(* CODESYS project Jacomex.project

Project tree, tasks and I/O mapping:
  IIoT_MQTT : XV300, Eaton Automation, version 3.5.19.30
    application Application
      libraries: StringUtils, 3.5.18.0 (System); VisuDialogs, * (System); Web Socket Client SL, 1.9.0.0 (CODESYS); Net Base Services, 3.5.19.20 (3S - Smart Software Solutions GmbH); MQTT Client SL, 1.9.0.0 (CODESYS); Standard, 3.5.18.0 (System); SysTimeRtc, * (System); SysTypes2 Interfaces, * (System)
      task MainTask (cyclic, interval t#20ms, priority 1) calls PRG
      program PRG [CFC]
      visualisation Visualization
      text list QoSTextlist
      function TerminateString [ST]
      image pool ImagePool
      text list ModeTextList
      text list VersionTextList
      global variables GVL_MQTT
      function FC_DataInMessageContainer [ST]
      data type ReactorType
  text list GlobalTextList
  5ce3da45-db07-42e7-a21c-a00fff4ed8f6|C:\Users\a.werner\Documents\background.jpg
  5ce3da45-db07-42e7-a21c-a00fff4ed8f6|C:\Users\a.werner\Documents\background.jpg
*)

// IIoT_MQTT/Application/ReactorType
{attribute 'qualified_only'}
TYPE ReactorType :
(
	O2 		:= 1,
	H2O 	:= 2,
	Both 	:= 3
)BYTE;
END_TYPE

// IIoT_MQTT/Application/GVL_MQTT
VAR_GLOBAL
	aValueData		:	ARRAY[1..20] OF DINT;		// Value data to transmit
	aTextData		:	ARRAY[1..20] OF STRING;		// Text data to transmit
	aBoolData		:	ARRAY[1..100] OF BOOL;		// Boolean data to transmit (Settings/Alarms/Triggers)
END_VAR

// IIoT_MQTT/Application/PRG
// MQTT Client with visualization
PROGRAM PRG
VAR
	//mqttClient 				: MQTT.MQTTClient; 								// Function block to establish a connection to a MQTT broker
	mqttPublisher 			: MQTT.MQTTPublish; 							// Function block to publish MQTT messages
	mqttPublisher2 			: MQTT.MQTTPublish; 							// Function block to publish MQTT messages
	mqttSubscriber 			: MQTT.MQTTSubscribe; 							// Function block to subscribe MQTT topics
	mqttSubscriber2 		: MQTT.MQTTSubscribe; 							// Function block to subscribe MQTT topics
	sHostname 				: STRING(255) 	:= 'mqtts-jacomex.ingelink.dev';//'broker.hivemq.com'; 				// Hostname or ip address or URL (for WebSockets: ws:// or wss://)
	wsUsername				: WSTRING 		:= "wildcard0";
	wsPassword				: WSTRING 		:= "f6eec544dc19429";
	uiPort 					: UINT 			:= 42226; 						// Port of the MQTT broker
	wsPublishTopic 			: WSTRING(1024) := "poly/in/1/0/5169/data"; 							// Topic to publish a message
	wsPublishTopic2 		: WSTRING(1024) := ""; 							// Topic to publish a message
	sWillMessage 			: STRING(1024); 								// The last will message
	abyPublishMessage 		: ARRAY [1..28] OF BYTE; 						// The messsage to publish
	sPublishMessage2 		: STRING(1024) := ''; 							// The messsage to publish 
	rsPub1Error				: RS; 											// Helper to publisher state
	rsPub1Done				: RS; 											// Helper to publisher state
	rsPub2Error				: RS; 											// Helper to publisher state
	rsPub2Done				: RS; 											// Helper to publisher state
	eCommunicationMode 		: MQTT.COMMUNICATION_MODE := MQTT.COMMUNICATION_MODE.TCP; // Communication mode: TCP/IP or WebSockets
	eMQTTVersion 			: MQTT.MQTT_VERSION := MQTT.MQTT_VERSION.V3_1_1; // The MQTT protocol version
	uiKeepAlive				: UINT 		:= 60;	
	sClientID				: STRING 	:= 'wildcard0';
	xCleanSession			: BOOL 		:= TRUE;
	

	
	// If you want to use client certificates, you can configure the connection via the TLS context.	
	 _sCommonName : STRING := 'MyXV303'; // CN of the certificate (common name). 
	 _sCipherList : NBS.CIPHER_LIST := STRUCT(psList := ADR('HIGH'), udiSize := 5); // Cipher string see https://www.openssl.org/docs/man1.1.1/man1/ciphers.html
	 _ciDefaultCertInfo : NBS.CERT_INFO := (psInfo := ADR(_sCommonName), udiSize := SIZEOF(_sCommonName)); // CN of the certificate (common name)

	 _tlsContext : NBS.TLSContext := (	sUseCaseName := _sCommonName, // A certificate is stored in the certificate store with the use case name. You can choose any name. Here we use the common name.
										ePurpose := NBS.PURPOSE.CLIENT_SIDE, // For client certificates set this to NBS.PURPOSE.CLIENT_SIDE
										sTLSVersion := '1.2', // The TLS version
										sCipherList := _sCipherList, // Set the cipher list
										udiVerificationMode := 1, // 2 => Active Peer verification
										ciCertInfo := _ciDefaultCertInfo, // Set the cert info
										itfCertVerifer := 0); // 0 => No Verifier 
	 
	 mqttClient : MQTT.MQTTClient := (itfTLSCOntext := _tlsContext);
    //
	// You can use the method TLSContext.SetInitialValue to set the context while runtime and set the context via the input itfTLSCOntext of the client FB.
	
	dwUuid: DWORD:= 5169;
	xFillingSolenoidValve: BOOL:=TRUE;
	wOxygenValue: WORD := 1664;
	sProject: STRING(16) := 'Project';
	eReactorType: ReactorType:= ReactorType.Both;
END_VAR
VAR // added by the converter: edge detectors and wires of the graphical bodies
    _w1 : ANY;
END_VAR

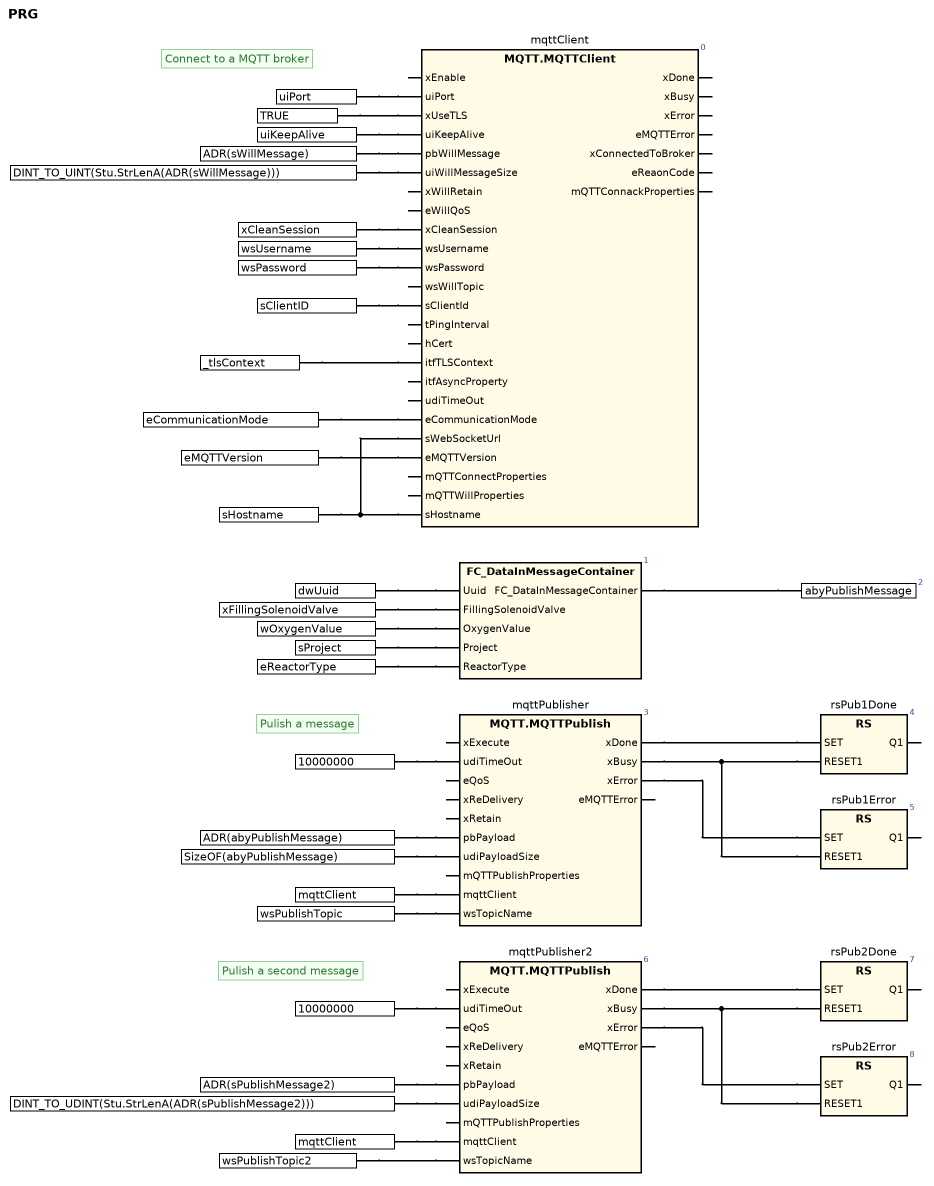
// Connect to a MQTT broker
mqttClient(
    uiPort := uiPort,
    xUseTLS := TRUE,
    uiKeepAlive := uiKeepAlive,
    pbWillMessage := ADR(sWillMessage),
    uiWillMessageSize := DINT_TO_UINT(Stu.StrLenA(ADR(sWillMessage))),
    xCleanSession := xCleanSession,
    wsUsername := wsUsername,
    wsPassword := wsPassword,
    sClientId := sClientID,
    itfTLSContext := _tlsContext,
    eCommunicationMode := eCommunicationMode,
    sWebSocketUrl := sHostname,
    eMQTTVersion := eMQTTVersion,
    sHostname := sHostname); // MQTT.MQTTClient
_w1 := FC_DataInMessageContainer(Uuid := dwUuid, FillingSolenoidValve := xFillingSolenoidValve, OxygenValue := wOxygenValue, Project := sProject, ReactorType := eReactorType);
abyPublishMessage := _w1;
// Pulish a message
mqttPublisher(
    udiTimeOut := 10000000,
    pbPayload := ADR(abyPublishMessage),
    udiPayloadSize := SizeOF(abyPublishMessage),
    mqttClient := mqttClient,
    wsTopicName := wsPublishTopic); // MQTT.MQTTPublish
rsPub1Done(SET := mqttPublisher.xDone, RESET1 := mqttPublisher.xBusy); // RS
rsPub1Error(SET := mqttPublisher.xError, RESET1 := mqttPublisher.xBusy); // RS
// Pulish a second message
mqttPublisher2(
    udiTimeOut := 10000000,
    pbPayload := ADR(sPublishMessage2),
    udiPayloadSize := DINT_TO_UDINT(Stu.StrLenA(ADR(sPublishMessage2))),
    mqttClient := mqttClient,
    wsTopicName := wsPublishTopic2); // MQTT.MQTTPublish
rsPub2Done(SET := mqttPublisher2.xDone, RESET1 := mqttPublisher2.xBusy); // RS
rsPub2Error(SET := mqttPublisher2.xError, RESET1 := mqttPublisher2.xBusy); // RS

END_PROGRAM

// IIoT_MQTT/Application/FC_DataInMessageContainer
FUNCTION FC_DataInMessageContainer : ARRAY [1..28] OF BYTE;
VAR_INPUT
	Uuid 					: DWORD; // hexa 4 
	FillingSolenoidValve 	: BOOL; // 1 
	OxygenValue  			: WORD; 		//Short (multiplié par 100) 2 
	Project 				: STRING(16); 
	ReactorType 			: ReactorType; 	// Enum 1
END_VAR
VAR
	_Result					: RTS_IEC_RESULT;
	_dwUtcTime				: DWORD;
	_dwLocalTime 			: DWORD;
	_dtLocalTime 			: DT;
END_VAR

//Copy UUID to Payload
FC_DataInMessageContainer[1] := UUID.%B0;
FC_DataInMessageContainer[2] := UUID.%B1;
FC_DataInMessageContainer[3] := UUID.%B2;
FC_DataInMessageContainer[4] := UUID.%B3;
//Create timespamp and copy to Payload
_dwUtcTime := SysTimeRtcGet(pResult:= _Result);
_Result := SysTimeRtcConvertUtcToLocal(dwTimestampUtc:= _dwUtcTime, pdwTimestampLocal:= _dwLocalTime);
_dtLocalTime := DWORD_TO_DT (_dwLocalTime);
FC_DataInMessageContainer[5] := _dwLocalTime.%B0;
FC_DataInMessageContainer[6] := _dwLocalTime.%B1;
FC_DataInMessageContainer[7] := _dwLocalTime.%B2;
FC_DataInMessageContainer[8] := _dwLocalTime.%B3;
//Copy FillingSolenoidValve to Payload
FC_DataInMessageContainer[9] := BOOL_TO_BYTE(FillingSolenoidValve);
//Copy OxygenValue to Payload
FC_DataInMessageContainer[10] := OxygenValue.%B0;
FC_DataInMessageContainer[11] := OxygenValue.%B1;
//Copy Project to Payload
FC_DataInMessageContainer[12] := Project[15];
FC_DataInMessageContainer[13] := Project[14];
FC_DataInMessageContainer[14] := Project[13];
FC_DataInMessageContainer[15] := Project[12];
FC_DataInMessageContainer[16] := Project[11];
FC_DataInMessageContainer[17] := Project[10];
FC_DataInMessageContainer[18] := Project[9];
FC_DataInMessageContainer[19] := Project[8];
FC_DataInMessageContainer[20] := Project[7];
FC_DataInMessageContainer[21] := Project[6];
FC_DataInMessageContainer[22] := Project[5];
FC_DataInMessageContainer[23] := Project[4];
FC_DataInMessageContainer[24] := Project[3];
FC_DataInMessageContainer[25] := Project[2];
FC_DataInMessageContainer[26] := Project[1];
FC_DataInMessageContainer[27] := Project[0];
//Copy ReactorType to Payload
FC_DataInMessageContainer[28] := ReactorType;

END_FUNCTION

// IIoT_MQTT/Application/TerminateString
// Terminates the STRING psIn at position udiLength
FUNCTION TerminateString : BOOL
VAR_INPUT
	psIn : POINTER TO BYTE; // Pointer to STRING
	udiLength : UDINT; // Length of psIn
END_VAR
VAR
END_VAR

psIn[udiLength] := 0;
TerminateString := TRUE;

END_FUNCTION

// IIoT_MQTT/Application/Visualization
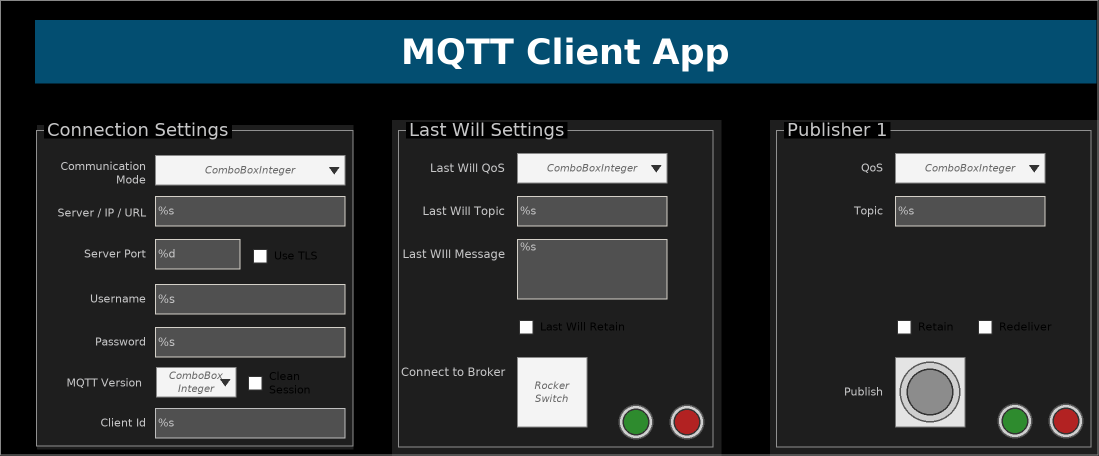
VISUALIZATION Visualization  // 1099x456
    Rectangle (37,125 316x324)
    Rectangle (392,120 329x336)
    GroupBox (398,122 315x325), "Last Will Settings"
        ComboBoxInteger (119,31 150x30), variable: PRG.mqttClient.eWillQoS, text list: 'QoSTextlist'
        Lamp1 (218,280 40x40), variable: PRG.mqttClient.xConnectedToBroker, style: Lamp-Lamp1-Green
        Lamp1 (269,280 40x40), variable: PRG.mqttClient.xError, style: Lamp-Lamp1-Red
    Label (408,153 100x30), "Last Will QoS"
    Textfield (517,196 150x30), "%s", text variable: PRG.mqttClient.wsWillTopic
        OnMouseClick: write the text variable via Default
    Label (408,196 100x30), "Last Will Topic"
    Textfield (517,239 150x60), "%s", text variable: PRG.sWillMessage
        OnMouseClick: write the text variable via Default
    Label (408,239 100x30), "Last WIll Message"
    Checkbox (517,312 150x30), "Last Will Retain", variable: PRG.mqttClient.xWillRetain
    Label (408,357 100x30), "Connect to Broker"
    RockerSwitch (517,357 70x70), variable: PRG.mqttClient.xEnable, behaviour: TOGGLE, style: Switch-RockerSwitch-Gray
    Rectangle (770,120 329x336)
    GroupBox (776,122 315x325), "Publisher 1"
    ComboBoxInteger (895,153 150x30), variable: PRG.mqttPublisher.eQoS, text list: 'QoSTextlist'
    Label (786,153 100x30), "QoS"
    Textfield (895,196 150x30), "%s", text variable: PRG.wsPublishTopic
        OnMouseClick: write the text variable via Default
    Label (786,196 100x30), "Topic"
    Checkbox (895,312 79x30), "Retain", variable: PRG.mqttPublisher.xRetain
    Checkbox (976,312 97x30), "Redeliver", variable: PRG.mqttPublisher.xReDelivery
    PushSwitch (895,357 70x70), variable: PRG.mqttPublisher.xExecute, input disabled if: NOT PRG.mqttClient.xConnectedToBroker, behaviour: TAP, style: Switch-PushSwitch-Gray
    Label (786,377 100x30), "Publish"
    Lamp1 (995,401 40x40), variable: PRG.rsPub1Done.Q1, style: Lamp-Lamp1-Green
    Lamp1 (1046,401 40x40), variable: PRG.rsPub1Error.Q1, style: Lamp-Lamp1-Red
    GroupBox (36,122 317x324), "Connection Settings"
        ComboBoxInteger (119,33 190x30), variable: PRG.eCommunicationMode, text list: 'ModeTextList'
        Label (-23,32 136x38), "Communication Mode"
        Textfield (119,74 190x30), "%s", text variable: PRG.sHostname
            OnMouseClick: write the text variable via Default
        Label (13,117 100x30), "Server Port", invisible if: PRG.eCommunicationMode = MQTT.COMMUNICATION_MODE.WEB_SOCKET
        Label (13,286 100x30), "Client Id"
        Textfield (119,286 190x30), "%s", text variable: PRG.mqttClient.sClientId
            OnMouseClick: write the text variable via Default
        Label (13,205 100x30), "Password"
        Textfield (119,205 190x30), "%s", text variable: PRG.mqttClient.wsPassword
            OnMouseClick: write the text variable via Default
        Label (13,162 100x30), "Username"
        Textfield (119,162 190x30), "%s", text variable: PRG.mqttClient.wsUsername
            OnMouseClick: write the text variable via Default
        Textfield (119,117 85x30), "%d", text variable: PRG.uiPort, invisible if: PRG.eCommunicationMode = MQTT.COMMUNICATION_MODE.WEB_SOCKET
            OnMouseClick: write the text variable via Default
        Label (-12,76 125x30), "Server / IP / URL"
        Checkbox (215,119 75x30), "Use TLS", variable: PRG.mqttClient.xUseTLS, invisible if: PRG.eCommunicationMode = MQTT.COMMUNICATION_MODE.WEB_SOCKET
        ComboBoxInteger (120,245 80x30), variable: PRG.eMQTTVersion, text list: 'VersionTextList'
        Label (23,246 86x30), "MQTT Version"
        Checkbox (210,246 103x30), "Clean Session", variable: PRG.mqttClient.xCleanSession
    Rectangle (35,20 1061x63), "MQTT Client App"
END_VISUALIZATION

(* text list QoSTextlist (id | default)
  0 | QoS 0
  1 | QoS 1
  2 | QoS 2
   |  *)

(* text list ModeTextList (id | default)
  0 | TCP/IP
  1 | WebSocket
   |  *)

(* text list VersionTextList (id | default)
  0 | 3.1.1
  1 | 5.0
   |  *)
